FUNCTION Celsius_To_Fahrenheit : REAL
VAR_INPUT
	fCelsius : REAL;
END_VAR
VAR
// scratch pad where program variables are stored.
END_VAR

Celsius_To_Fahrenheit := fCelsius * 1.8 + 32.0;

END_FUNCTION

(* stored: Version 1.1.0.1, ProductVersion 3.1.4024.11
   POU Celsius_To_Fahrenheit: Id {90345588-d78c-4f6d-a4a3-670fbd7f85e5}, SpecialFunc None *)
